// TwinCAT 3 PLC project Program_2
// ProgramVersion: 3.1.4024.0
// libraries:
//   Inputs and outputs, * (MyCompany AB)
//   Tc2_Standard, * (Beckhoff Automation GmbH)
//   Tc2_System, * (Beckhoff Automation GmbH)
//   Tc3_Module, * (Beckhoff Automation GmbH)
// project tree:
//   / PlcTask.TcTTO
//   POUs/ FB_TestFunctionBlock.TcPOU, MAIN.TcPOU
// real-time tasks:
//   TASK PlcTask: cycle T#10ms, priority 20, ADS port 350

CONFIGURATION Program_2
    RESOURCE PLC ON TwinCAT3
        TASK PlcTask(INTERVAL := T#10ms, PRIORITY := 20);
        PROGRAM MAIN WITH PlcTask : MAIN;
    END_RESOURCE
END_CONFIGURATION

// ---- POUs/MAIN.TcPOU
PROGRAM MAIN
VAR
	fbFactorial : IO.Factorial;
	fbFactorial_2 : IO.Factorial;
END_VAR

fbFactorial(); 
fbFactorial_2();

END_PROGRAM

// ---- POUs/FB_TestFunctionBlock.TcPOU
FUNCTION_BLOCK FB_TestFunctionBlock
VAR
	nCounter : LINT;
END_VAR

nCounter := nCounter + 1;

END_FUNCTION_BLOCK
